/// Enumeration of all plant components
TYPE E_Component :
(
	/// component not set
	eComponent_none := 0,

	/// component max index (keep @ last)
	eComponent_nMaxIdx
);
END_TYPE

(* stored: Version 1.1.0.1, ProductVersion 3.1.4024.11
   DUT E_Component: Id {781dfb0a-629c-4aa9-8271-3df78a05904a} *)
